// TIA Portal V17 export
// export: Created 2026-04-13T11:12:42.1145092Z, ExportSetting WithDefaults, DisplayName Totally Integrated Automation Portal, DisplayVersion V17 Update 4, DisplayName TIA Portal Openness, DisplayVersion V17 Update 4, DisplayName TIA Portal Version Control Interface, DisplayVersion V17, DisplayName SINAMICS Startdrive Advanced, DisplayVersion V17, DisplayName SINAMICS Startdrive G130, G150, S120, S150, SINAMICS MV, S210, DisplayVersion V17, DisplayName SINAMICS Startdrive G110M, G120, G120C, G120D, G120P, G115D, DisplayVersion V17, DisplayName STEP 7 Professional, DisplayVersion V17 Update 4, DisplayName STEP 7 Safety, DisplayVersion V17, DisplayName WinCC Professional, DisplayVersion V17 Update 4
FUNCTION_BLOCK "步段延迟"   // FB65, SCL
{ S7_Optimized_Access := 'TRUE' }
VERSION : 0.1
// stored: AutoNumber true, IsIECCheckEnabled false, IsRetainMemResEnabled false, MemoryReserve 100, SetENOAutomatically false, UDAEnableTagReadback false
   VAR_INPUT
      YC延迟设定时间 : Real := 50.0;   // 设定延迟时间
   END_VAR
   VAR_IN_OUT
      "AND" : Bool;   // 延迟的条件
      Q : Bool;   // 延迟时间到达后执行的动作
      YX运行时间 : Real;   // 显示时钟时间
   END_VAR
   VAR
      T1S : TON_TIME;   // 1秒脉冲
   END_VAR
BEGIN
   IF #T1S.Q AND #YX运行时间 < #YC延迟设定时间 AND #AND THEN
       #YX运行时间 := #YX运行时间 + 1;
   END_IF;

   IF #YX运行时间 >= #YC延迟设定时间 THEN
       #Q := 1;
   END_IF;

   (* IF NOT #AND THEN
       #YX运行时间 := 0;
       #Q := 0;
   END_IF; *)

   #T1S(IN := NOT #T1S.Q,
          PT := T#1S);
END_FUNCTION_BLOCK
